// TwinCAT 3 PLC project MC3_Multi_IPC1
// ProgramVersion: 3.1.4026.13
// libraries:
//   Tc2_EtherCAT, * (Beckhoff Automation GmbH)
//   Tc2_Standard, * (Beckhoff Automation GmbH)
//   Tc2_System, * (Beckhoff Automation GmbH)
//   Tc2_Utilities, * (Beckhoff Automation GmbH)
//   Tc3_EventLogger, * (Beckhoff Automation GmbH)
//   Tc3_Mc3PlanarMotion, * (Beckhoff Automation GmbH)
//   Tc3_Module, * (Beckhoff Automation GmbH)
//   Tc3_Physics, * (Beckhoff Automation GmbH)
//   Tc3_XL_Motion, * (Beckhoff Automation GmbH)
//   Tc3_XtsInterface,newest,Beckhoff Automation GmbH
// project tree:
//   DUTs/ E_EcState.TcDUT (not stored), E_MergeMode.TcDUT (not stored), E_MergeType.TcDUT (not stored), E_SwitchOpMode.TcDUT (not stored), E_TrackNum.TcDUT, MoverSort.TcDUT (not stored), ST_Color_Code.TcDUT (not stored), ST_DivertConfig.TcDUT (not stored), ST_ExpMoverStatus.TcDUT (not stored), ST_MergeConfig.TcDUT (not stored), ST_MoverConfig.TcDUT (not stored), ST_PlanarTrackConfig.TcDUT (not stored), ST_SectorConfig.TcDUT (not stored), ST_ShortcutConfig.TcDUT (not stored), ST_StaticSectorStatus.TcDUT (not stored), ST_SwitchConfig.TcDUT (not stored), ST_SwitchStatus.TcDUT (not stored), ST_TrackConfig.TcDUT (not stored)
//   GVLs/ GVL_DataExchange.TcGVL, GVL_MC.TcGVL
//   / PlcTask.TcTTO (not stored)
//   POUs/ FB_PWM.TcPOU, FB_TrackObject.TcPOU, IsBetween.TcPOU (not stored), MAIN_S1.TcPOU, F_GetTrackEnum.TcPOU (not stored)
//   XlMover/DUTs/ DUT.TcDUT (not stored), ST_MoverInfo.TcDUT (not stored), ST_MoverOnTrackInfo.TcDUT
//   XlMover/ITFs/ I_Mover.TcIO
//   XlMover/POUs/ FB_Mover.TcPOU

// ---- DUTs/E_TrackNum.TcDUT
TYPE E_TrackNum :
{attribute 'qualified_only'}
{attribute 'strict'}
	(
	MainStart 	:= 1,	
	Big 		:= 2,
	MainEnd		:= 3,
	Small 		:= 4);	
END_TYPE

// ---- XlMover/DUTs/ST_MoverOnTrackInfo.TcDUT
TYPE ST_MoverOnTrackInfo :
STRUCT
	TargetPosition 		: LREAL;
	TargetTrack 		: Otcid;
	Remainingdistance 	: LREAL;
	Gap 				: LREAL;
	LimitV 				: LREAL;
	LimitA 				: LREAL;
	LimitD 				: LREAL;
	LimitJ 				: LREAL;
	GapMode				: MC.MC_GAP_MODE_ON_TRACK;
	DynamicMode			: MC.MC_DYNAMIC_MODE_ON_TRACK;
	Movementtype		: MC.MC_MOVEMENT_TYPE_ON_TRACK;
	
END_STRUCT
END_TYPE

// ---- GVLs/GVL_DataExchange.TcGVL
{attribute 'qualified_only'}
VAR_GLOBAL
	Dynamics AT%Q*: ST_Dynamics;
	Reset : BOOL;
	Run: BOOL;
	SafetyInRun : BOOL; 
	
	aMoverInfos : ARRAY[1..nNumMovers] OF ST_MoverInfo;
	
	
END_VAR

// ---- GVLs/GVL_MC.TcGVL

VAR_GLOBAL CONSTANT
	nNumMovers			: UINT := 12;
	nNumTracks			: UINT := 4;
	XtsShortcutOid				: otcid := 16#01010490 ;
	XtsOutterLoopOid 			: otcid := 16#01010480;
	
	fMagnetEntry : LREAL := 1766; //PLEASE ENTER THE MAGNET ENTRY!!!
	fMagnetExit : LREAL := 2332; //PLEASE ENTER THE MAGNET EXIT!!!
	
    standardAccel : LREAL := 4000; 
    standardDecel : LREAL :=4000; 
    standardJerk : LREAL := 16000; 

END_VAR
VAR_GLOBAL PERSISTENT
	nNumActiveMovers	: UINT := 1;
END_VAR	
VAR_GLOBAL
	

	fbXtsEnvironment			: 	FB_XtsEnvironment;
	ipXtsProcessingUnit			:   I_XtsProcessingUnit1;
	cmdFeedback					: 	XtsCommandFeedback;
	buffer						:   BYTE;
	
	fbMover						:	ARRAY[1..GVL_MC.nNumMovers] OF FB_Mover;
	iMover						:	ARRAY[1..GVL_MC.nNumMovers] OF I_Mover;
	aDynamics					:  	DynamicConstraint_PathXY;
	Feedback 					:	ARRAY[1..GVL_MC.nNumMovers] OF MC_PlanarFeedback;
	TrackFeedback 				:	ARRAY[1..GVL_MC.nNumTracks] OF MC_PlanarFeedback;
	aMcTracks					:	ARRAY[1..GVL_MC.nNumTracks] OF MC_PlanarTrack;
	ExitSystem 					: 	MC_PlanarTrackConnectionOut;
	EnterSystem 				:	MC_PlanarTrackConnectionIn;	
	Mover						:	ARRAY[0..GVL_MC.nNumMovers] OF MoverSort;
	defaultGap					:	LREAL := 900.0;
	SafetyOK			 AT %I* :	BOOL;
END_VAR

// ---- XlMover/ITFs/I_Mover.TcIO

INTERFACE I_Mover

METHOD CycleUpdate : BOOL
VAR_INPUT
END_VAR
END_METHOD

PROPERTY distToEndOfTrack : Lreal
GET
END_GET
END_PROPERTY

METHOD Init : BOOL
VAR_INPUT
	XtsMover:  I_XtsXlMover1;
	XtsProcessingUnit :  I_XtsProcessingUnit1;
END_VAR
END_METHOD

METHOD JoinNearestTrack : BOOL


VAR

END_VAR
END_METHOD

METHOD LeaveSystemAt : BOOL
VAR_INPUT
	ConnectionOut: REFERENCE TO MC_PlanarTrackConnectionOut;	
	gap : LREAL; 		
END_VAR
END_METHOD

METHOD MoveOnTrack : BOOL
VAR_INPUT
	track: REFERENCE TO MC_PlanarTrack;	
	targetPos: LREAL;
	gap : LREAL; 

END_VAR
END_METHOD

PROPERTY MoverStopped : BOOL
GET
END_GET
SET
END_SET
END_PROPERTY

PROPERTY P_Dynamics : REFERENCE TO DynamicConstraint_PathXY;
GET
END_GET
END_PROPERTY

PROPERTY P_IsInitialized : bool
GET
END_GET
END_PROPERTY

PROPERTY P_MoverOTCID : OTCID
GET
END_GET
SET
END_SET
END_PROPERTY

PROPERTY P_PlanarFeedback : REFERENCE TO MC_PlanarFeedback
GET
END_GET
END_PROPERTY

PROPERTY P_PlanarMover :   REFERENCE TO  MC_PlanarMover
GET
END_GET
END_PROPERTY

PROPERTY P_SyncFeedback :  REFERENCE TO MC_PlanarFeedbackGearInPosOnTrackWithMasterMover
GET
END_GET
END_PROPERTY

PROPERTY P_TargetTrack : UDINT
GET
END_GET
SET
END_SET
END_PROPERTY

PROPERTY Rework : BOOL
GET
END_GET
SET
END_SET
END_PROPERTY

METHOD SyncToOtherMover : Bool
VAR_INPUT
	masterSyncPos : LREAL; // Position on the master track
	followerSyncPos : LREAL; // position on the follower track
	PlanarMoverToFollow: REFERENCE TO Tc3_Mc3PlanarMotion.MC_PlanarMover;
	masterTrack : REFERENCE TO Tc3_Mc3PlanarMotion.MC_PlanarTrack; 
	followerTrack : REFERENCE TO Tc3_Mc3PlanarMotion.MC_PlanarTrack; 
	velo :  REFERENCE TO LREAL; 
END_VAR
END_METHOD

METHOD  UpdateXtsTrack
VAR_INPUT
END_VAR
VAR

END_VAR
END_METHOD

PROPERTY XlProcessingUnit : I_XtsProcessingUnit1
GET
END_GET
END_PROPERTY

PROPERTY XtsComFeed : REFERENCE TO  XtsCommandFeedback
GET
END_GET
END_PROPERTY

PROPERTY XtsXlMover :  I_XtsXlMover1
GET
END_GET
END_PROPERTY

END_INTERFACE

// ---- XlMover/POUs/FB_Mover.TcPOU
{attribute 'no_assign'}
FUNCTION_BLOCK FB_Mover IMPLEMENTS I_Mover
VAR_INPUT
END_VAR
VAR_OUTPUT
END_VAR
VAR
	_bIsInitialized: BOOL;	

	fbPlanarMover : MC_PlanarMover;
	fbPlanarFeedback: MC_PlanarFeedback;
	trackTrail: MC_PlanarTrackTrail;
	SyncMoverFeedback: Tc3_Mc3PlanarMotion.MC_PlanarFeedbackGearInPosOnTrackWithMasterMover;
	
	_GearInOptions: Tc3_Mc3PlanarMotion.ST_GearInPosOnTrackWithMasterMoverOptions;
	_stMoveOnTrackOptions: ST_MoveOnTrackOptions;
	_stLeaveSystemAtOptions : ST_LeaveSystemAtOptions;
	
	_syncTrail : MC_PlanarTrackTrail;
	
	CmdFeedback :  XtsCommandFeedback;
	ipXtsMover:   I_XtsXlMover1;
	ipXtsProcessingUnit:  I_XtsProcessingUnit1;

	_stMoverInfos : ST_MoverInfo;	
	_stMoverOnTrackInfos : MC_MOVER_ON_TRACK_INFORMATION;

	_nextMcTrackOid: OTCID;
	_stDynamics: DynamicConstraint_PathXY;
	_TargetTrack : UDINT;
	_ReWork : BOOL;
	_partConfig: UINT;
	_InSync :BOOL; 
	_PositionOnTrack : LREAL;
	_Track : OTCID; 
	_distToEndOfTrack : LREAL;

	fbResult						: FB_TcMessage;
	_ipComObject					: ITComObject;
	PID_OnTrackInfos				: PTCID := 16#05030180;
	bInit 							: BOOL;
END_VAR



METHOD CycleUpdate : BOOL
VAR_INPUT
END_VAR

VAR_INST
	_trackEnum: e_TrackNum;

END_VAR
IF NOT _bIsInitialized THEN
	RETURN;
END_IF

fbPlanarMover.GetTrackTrailInformation(trackTrail);
_PositionOnTrack := fbPlanarMover.MCTOPLC.SETONTRACK.SetPos;
IF fbPlanarMover.MCTOPLC.SETONTRACK.TrackOID<>0 THEN 
	_Track := fbPlanarMover.MCTOPLC.SETONTRACK.TrackOID;
	_trackEnum := F_GetTrackEnum(fbPlanarMover.MCTOPLC.SETONTRACK.TrackOID); 
	_distToEndOfTrack := GVL_Mc.aMCTracks[_trackEnum].GetLength()-_PositionOnTrack;
END_IF

fbPlanarMover.Update();
fbPlanarFeedback.Update();
SyncMoverFeedback.Update();

_stMoverinfos.MoverOtcid :=TO_STRING(fbPlanarMover.MCTOPLC.STD.MoverOID) ;
_stMoverinfos.IsActive := ipXtsMover.GetIsActive(0);
_stMoverinfos.ActPos :=  ipXtsMover.GetPositionInfo_trackPosition(0);
_stMoverinfos.ActVelo := fbPlanarMover.MCTOPLC.SETONTRACK.SetVelo;
_stMoverinfos.IsVirtuell := ipXtsMover.GetIsVirtualFeedbackEnabled(0);
_stMoverinfos.Positition :=	fbPlanarMover.MCTOPLC.SETONTRACK.SetPos;
_stMoverinfos.Track := TO_STRING(_trackEnum);
_stMoverinfos.Error := fbPlanarMover.Error;
_stMoverinfos.ErrorID := fbPlanarMover.ErrorId;
_stMoverinfos.PlanarMoverCommandMode :=  TO_STRING(fbPlanarMover.MCTOPLC.STD.CommandMode);
_stMoverinfos.State :=  TO_STRING(fbPlanarMover.MCTOPLC.STD.State);
_stMoverinfos.Gap := _stMoverOnTrackInfos.Gap;
_stMoverinfos.LimitAcc := _stMoverOnTrackInfos.LimitA;
_stMoverinfos.LimitDec := _stMoverOnTrackInfos.LimitD;
_stMoverinfos.LimitJerk := _stMoverOnTrackInfos.LimitJ;
_stMoverinfos.LimitVelo := _stMoverOnTrackInfos.LimitV;
_stMoverinfos.TargetTrackPosition := _stMoverOnTrackInfos.TargetPosition;
_stMoverinfos.TargetTrack := _stMoverOnTrackInfos.TargetTrack;
_stMoverinfos.RemainingDistance := _stMoverOnTrackInfos.Remainingdistance;




UpdateXtsTrack();
GetOnTrackInfos() ;
END_METHOD

PROPERTY distToEndOfTrack : Lreal
GET
distToEndOfTrack := _distToEndOfTrack;
END_GET
END_PROPERTY

METHOD GetComObject : BOOL
VAR_INPUT
	nObjectId: OTCID;
END_VAR
IF FW_ObjMgr_GetObjectInstance(	oid		:= nObjectId, 
								iid		:= TC_GLOBAL_IID_LIST.IID_ITComObject, 
								pipUnk	:= ADR(_ipComObject)) = 0
THEN
	GetComObject := TRUE;
END_IF
END_METHOD

METHOD GetOnTrackInfos : BOOL
VAR
	nData 			: UDINT := SIZEOF(MC_MOVER_ON_TRACK_INFORMATION);
	pData 			: PVOID := ADR(MC_MOVER_ON_TRACK_INFORMATION);
	stEventEntry	: TcEventEntry;
	pstEventEntry	: REFERENCE TO TcEventEntry REF= stEventEntry;
END_VAR
VAR_INST
	hResult : HRESULT;
	bError : BOOL;
END_VAR
bError := FALSE;

IF _ipComObject <> 0 THEN 
	 hResult := 	_ipComObject.TcgetObjPara(		pid := PID_OnTrackInfos,
													nData := nData,
													pData := pData,
													pgp := 0); 	
	IF hResult = 0 THEN
		GetOnTrackInfos := TRUE;
ELSE
	HRESULTAdsErr_TO_TcEventEntry(hResult,stEventEntry);
	IF NOT fbResult.EqualsToEventEntryEx( stOther := stEventEntry) THEN
		fbResult.CreateEx(stEventEntry, 0);
		fbResult.Send(0);
		fbResult.Release();
	END_IF
		bError := TRUE;
	END_IF							
END_IF
END_METHOD

METHOD Init : BOOL
VAR_INPUT

	XtsMover:   I_XtsXlMover1;
	XtsProcessingUnit :  I_XtsProcessingUnit1;
END_VAR



ipXtsMover:= XtsMover;
ipXtsProcessingUnit :=  XtsProcessingUnit;

_stMoveOnTrackOptions.direction := MC_Direction.mcDirectionPositive;
_stMoveOnTrackOptions.gapMode := MC_GAP_MODE_ON_TRACK.Fast1D;
_stMoveOnTrackOptions.gap:= 800;

_syncTrail.AddTrack(track:= GVL_Mc.aMCTracks[E_TrackNum.Small]); 
_syncTrail.AddTrack(track:= GVL_Mc.aMCTracks[E_TrackNum.MainStart]); 


//_stDynamics.SetValuesVADJ(500, 4000, 4000, 10000);




	_bIsInitialized := TRUE;
	Init := TRUE;

IF NOT bInit THEN
	IF GetComObject(nObjectId:=fbPlanarMover.MCTOPLC.STD.MoverOID) THEN
		bInit:=TRUE;
	END_IF
	RETURN;
END_IF
END_METHOD

METHOD JoinNearestTrack : BOOL


VAR_INST
	nForCounter: UINT;
	mcTrackOid: OTCID;
	partOid: OTCID;
	cmdFeedback					: 	XtsCommandFeedback;
	objectInfo: PlanarObjectInfo;
END_VAR
partOid := ipXtsMover.GetPositionInfo_partObjectId(cmdFeedback);

IF partOid = 0 THEN
	RETURN;
END_IF

IF cmdFeedback.IsDone THEN
	mcTrackOid := ipXtsProcessingUnit.XlPartWithOid(partOid, cmdFeedback).GetMcTrackOid(cmdFeedback);
	
	FOR nForCounter := 1 TO GVL_MC.nNumTracks DO
		objectInfo := GVL_MC.aMcTracks[nForCounter].GetPlanarObjectInfo();
		IF objectInfo.Id = mcTrackOid THEN
			fbPlanarMover.JoinTrack(fbPlanarFeedback, GVL_MC.aMcTracks[nForCounter], _stDynamics, 0); 
			RETURN;
		END_IF
	END_FOR
END_IF
END_METHOD

METHOD LeaveSystemAt : BOOL
VAR_INPUT
	ConnectionOut: REFERENCE TO MC_PlanarTrackConnectionOut;
	gap : LREAL; 
END_VAR
_stLeaveSystemAtOptions.gap := gap;
_stLeaveSystemAtOptions.gapMode := MC_GAP_MODE_ON_TRACK.Fast1D; 
_stLeaveSystemAtOptions.dynamicMode :=  MC_DYNAMIC_MODE_ON_TRACK.None;

fbPlanarMover.LeaveSystemAt(fbPlanarFeedback, ConnectionOut,  _stDynamics,_stLeaveSystemAtOptions);
END_METHOD

METHOD MoveOnTrack : BOOL
VAR_INPUT
	track: REFERENCE TO MC_PlanarTrack;	
	targetPos: LREAL;
	gap : LREAL; 
END_VAR
_stMoveonTrackOptions.gap := gap; 

fbPlanarMover.MoveOnTrack(
	commandFeedback:= fbPlanarFeedback, 
	targetTrack:= track, 
	targetPositionOnTrack:= targetPos, 
	constraint:= _stDynamics, 
	options:= _stMoveOnTrackOptions);
END_METHOD

PROPERTY MoverStopped : BOOL
GET
MoverStopped := (fbPlanarMover.MCTOPLC.SETONTRACK.SetVelo < 20);
END_GET
SET
END_SET
END_PROPERTY

PROPERTY P_Dynamics : REFERENCE TO DynamicConstraint_PathXY;
GET

P_Dynamics REF= _stDynamics;
END_GET
END_PROPERTY

PROPERTY P_IsInitialized : bool
GET
P_IsInitialized := _bIsInitialized;
END_GET
END_PROPERTY

PROPERTY P_MoveOnTrackOptions  : REFERENCE TO  ST_MoveOnTrackOptions
GET
P_MoveOnTrackOptions REF= _stMoveOnTrackOptions;
END_GET
END_PROPERTY

PROPERTY P_MoverInfos : REFERENCE TO ST_MoverInfo
GET
P_MoverInfos  REF= _stMoverInfos;
END_GET
END_PROPERTY

PROPERTY p_MoverOTCID : OTCID
GET
p_MoverOTCID := fbPlanarMover.MCTOPLC.STD.MoverOID;
END_GET
SET
END_SET
END_PROPERTY

PROPERTY P_PlanarFeedback : REFERENCE TO MC_PlanarFeedback
GET
P_PlanarFeedback REF= fbPlanarFeedback;
END_GET
END_PROPERTY

PROPERTY P_PlanarMover :   REFERENCE TO  MC_PlanarMover
GET
P_PlanarMover REF= fbPlanarMover;
END_GET
END_PROPERTY

PROPERTY P_SyncFeedback :  REFERENCE TO MC_PlanarFeedbackGearInPosOnTrackWithMasterMover
GET
P_SyncFeedback REF= SyncMoverFeedback;
END_GET
END_PROPERTY

PROPERTY P_TargetTrack : UDINT
GET
P_TargetTrack := _TargetTrack ;
END_GET
SET
_TargetTrack := P_TargetTrack;
END_SET
END_PROPERTY

PROPERTY Rework : BOOL
GET
Rework := _Rework;
END_GET
SET
_Rework := Rework;
END_SET
END_PROPERTY

METHOD SyncToOtherMover : BOOL
VAR_INPUT
	masterSyncPos : LREAL; // Position on the master track
	followerSyncPos : LREAL; // position on the follower track
	PlanarMoverToFollow: REFERENCE TO Tc3_Mc3PlanarMotion.MC_PlanarMover;
	masterTrack : REFERENCE TO Tc3_Mc3PlanarMotion.MC_PlanarTrack; 
	followerTrack : REFERENCE TO Tc3_Mc3PlanarMotion.MC_PlanarTrack; 
	velo : REFERENCE TO LREAL; 
END_VAR

VAR
	trail: Tc3_Mc3PlanarMotion.MC_PlanarTrackTrail;

END_VAR
_GearInOptions.allowedSlaveSyncDirections := MC_SYNC_DIRECTIONS.Positive; 
_GearInOptions.directionMasterSyncPosition := MC_DIRECTION.mcDirectionNonModulo; 
_GearInOptions.directionSlaveSyncPosition := MC_DIRECTION.mcDirectionNonModulo;  
_GearInOptions.followMover := FALSE; 
_GearInOptions.gap := 0; // elimnate gap funciton 
_GearInOptions.inSyncToleranceDistance :=0; 
_GearInOptions.moduloToleranceMasterSyncPosition := 0; 
_GearInOptions.moduloToleranceSlaveSyncPosition := 0;  
_stDynamics.V := velo; 

fbPlanarMover.GearInPosOnTrackWithMasterMover(
	commandFeedback:=  SyncMoverFeedback , 
	masterMover:= PlanarMoverToFollow , 
	trackTrail:= _syncTrail, // may need to give a trail maybe not
	masterSyncPosition:= masterSyncPos, 
	masterSyncPositionTrack:= MasterTrack , 
	slaveSyncPosition:= followerSyncPos, 
	slaveSyncPositionTrack:= followerTrack, 
	constraint:=_stDynamics , 
	options:=_GearInOptions );
END_METHOD

METHOD PUBLIC UpdateXtsTrack
VAR_INPUT
END_VAR
VAR_STAT
	nTrackCount: UINT;
	oid1: OTCID;
	oid2: OTCID;
	
	nForCounter: UINT;
	nPartConfigCount: UINT;
	
	partConfig1: OTCID;
	partConfig2: OTCID;
	
	mcTrackOid1: OTCID;
	mcTrackOid2: OTCID;
	trackOid: OTCID;
	
	nTrackTrailCount: UDINT;
	actTrackOid: OTCID;
	nIndexInTrail: UDINT;
END_VAR
nTrackTrailCount := trackTrail.TrackCount;
actTrackOid := fbPlanarMover.MCTOPLC.SETONTRACK.TrackOID;

IF nTrackTrailCount <= 1 THEN
	RETURN;
END_IF

FOR nForCounter := 1 TO UDINT_TO_UINT(nTrackTrailCount) DO
	oid1 := trackTrail.GetTrackOidAt(nForCounter);
	IF oid1 = actTrackOid THEN
		IF nForCounter < nTrackTrailCount THEN
			oid2 := trackTrail.GetTrackOidAt(nForCounter + 1);
			EXIT;
		ELSE
			RETURN; //last one ine track trail
		END_IF
	END_IF
END_FOR

IF oid2 = _nextMcTrackOid AND ipXtsMover.GetPositionInfo_partPosition(CmdFeedback) < 600 THEN //no change
	RETURN;
END_IF

nTrackCount := ipXtsProcessingUnit.TrackCount();

FOR nForCounter := 1 TO nTrackCount DO
	nPartConfigCount := ipXtsProcessingUnit.Track(nForCounter, CmdFeedback).PartConfigCount(); 
	
	IF nPartConfigCount >= 2  THEN
		partConfig1 := ipXtsProcessingUnit.Track(nForCounter, CmdFeedback).GetPartConfigOidAt(1, 0);
		partConfig2 := ipXtsProcessingUnit.Track(nForCounter, CmdFeedback).GetPartConfigOidAt(2, 0);
//
		
		IF partConfig1 = 0 OR partConfig2 = 0 THEN
			CONTINUE;
		END_IF
		
		mcTrackOid1 := ipXtsProcessingUnit.XlPartWithOid(partConfig1, CmdFeedback).GetMcTrackOid(0);
		mcTrackOid2 := ipXtsProcessingUnit.XlPartWithOid(partConfig2, CmdFeedback).GetMcTrackOid(0);
		IF mcTrackOid1 = oid1 AND mcTrackOid2 = oid2   THEN
			trackOid := ipXtsProcessingUnit.Track(nForCounter, CmdFeedback).GetObjectId();
			ipXtsMover.SetActiveTrackObjectId(trackOid, CmdFeedback);
			
			IF CmdFeedback.IsDone THEN
				_nextMcTrackOid := oid2;
			END_IF
			
			RETURN;
		END_IF
	END_IF
END_FOR
END_METHOD

PROPERTY XlProcessingUnit : I_XtsProcessingUnit1
GET
XlProcessingUnit := ipXtsProcessingUnit;
END_GET
END_PROPERTY

PROPERTY XtsComFeed : REFERENCE TO  XtsCommandFeedback
GET
XtsComFeed REF= CmdFeedback;
END_GET
END_PROPERTY

PROPERTY XtsXlMover : I_XtsXlMover1
GET
XtsXlMover := ipXtsMover;
END_GET
END_PROPERTY

END_FUNCTION_BLOCK

// ---- POUs/FB_PWM.TcPOU
FUNCTION_BLOCK FB_PWM
VAR_INPUT
	SafeetyOk : BOOL;
	Torque: INT;
END_VAR

VAR
  	ModuleState AT %I* : UINT;
	
 	Control AT %Q* :  UINT;
 	TargetTorque AT %Q*: INT; 	

 	State  : INT := 1;
 	PwmTimer : ton;
END_VAR

VAR_OUTPUT
	Ready : BOOL;
END_VAR


Ready := FALSE;
CASE State OF 

	1:
		IF SafeetyOk THEN
			State := 2;
		END_IF
	2: 
		Control := 6;
		IF ModuleState = 40 OR ModuleState = 33 THEN
			State := 5;
		END_IF
	5:
		Control := 128;
		IF ModuleState = 96 OR ModuleState = 33 OR ModuleState = 168 THEN
			State := 10;
		END_IF
	10:
		Control := 6;
		IF ModuleState = 33 THEN
			state := 15;
		END_IF	
	15:
		Control := 7;
		IF ModuleState = 35 OR ModuleState = 163 or ModuleState = 2083 THEN
			State := 20;
		END_IF	
	20:	
		Control := 15;
		IF ModuleState = 4135 OR ModuleState = 4263THEN
			state := 25;
		END_IF
	24:
	  //IF Torque = 0  THEN
			State := 25;
	//	END_IF	
		PwmTimer(in := FALSE,PT := T#30S);
	25:
		IF ModuleState = 40 THEN
			State := 5;
		END_IF
		Ready := TRUE;
		
		IF Torque > 0 THEN
			TargetTorque := Torque ;
		ELSIF Torque = 0 AND TargetTorque > 0  THEN	
			TargetTorque :=  TargetTorque - REAL_TO_INT((INT_TO_REAL(TargetTorque)*0.07));
		END_IF	
		
		PwmTimer(in := TargetTorque > 300,PT := T#30S);
		IF PwmTimer.Q  THEN
			PwmTimer(in := FALSE,PT := T#30S);
			State := 35;
		END_IF 
	35:
		IF TargetTorque >0 THEN
			TargetTorque := TargetTorque -4;
		ELSIF 	TargetTorque = 0  THEN
				State := 24;
		END_IF	

END_CASE

END_FUNCTION_BLOCK

// ---- POUs/FB_TrackObject.TcPOU
FUNCTION_BLOCK FB_TrackObject
// for a track/part this block keeps a list of the movers in order with their positions on a track

VAR_INPUT
	TrackID: OTCID;
	iMover	:REFERENCE TO ARRAY[1..nNumMovers] OF I_Mover;
	trackLength : LREAL;// this should be a loookup but I don't know how to look it up so I'm going to pass it externally 
END_VAR

VAR_OUTPUT
	bBusy: BOOL;
	bDone: BOOL;
	bError: BOOL;
	bInit: BOOL;
	ipResultMessage: I_TcMessage := fbResult;
	moverIDs : ARRAY[1..nNumMovers] OF UDINT;
END_VAR

VAR
	nNumMoversThisTrack: UDINT; //numberofMovers currently on this track
	nMoverList: ARRAY [1..nNumMovers] OF OTCID; //list of movers currently on the track 

	distToNextMover : ARRAY[1..nNumMovers] OF LREAL;  
END_VAR

VAR

	fbResult: FB_TcMessage;
	_ipComObject: ITComObject;
	PID_MOverList				: PTCID := 16#05030149;
	PID_NumMover				: PTCID := 16#050300C5;
END_VAR

IF NOT bInit THEN
	IF GetComObject(nObjectId:=TrackID) THEN
		bInit:=TRUE;
	END_IF
	RETURN;
END_IF

METHOD CyclicUpdate : BOOL
VAR_INPUT
END_VAR

VAR
	J: UDINT;
	I: UDINT;
END_VAR
IF bInit THEN 
	GetNumMovers(); 
	GetMoverList(); 
END_IF 
MEMSET(ADR(moverIDs),0,SIZEOF(moverIDs)); // have to clear the list 
FOR J := 1 TO nNumMoversThisTrack DO  
	FOR I := 1 TO nNumMovers DO  
		IF iMover[I].P_MoverOTCID = nMoverList[J] THEN 
			moverIDs[J] := I; 
		END_IF
	END_FOR
END_FOR
FOR I := 1 TO nNumMoversThisTrack DO 
	IF I <= nNumMoversThisTrack -1 THEN
		distToNextMover[I] := fbMover[moverIDs[I+1]].distToEndOfTrack - fbMover[moverIDs[I]].distToEndOfTrack;
	ELSIF I = nNumMoversThisTrack THEN
		distToNextMover[I] := trackLength - fbMover[moverIDs[I]].distToEndOfTrack;
	END_IF
END_FOR
END_METHOD

METHOD findMergePosition : BOOL
VAR_INPUT
	mergeSyncCommandPos : LREAL;
	spaceToMerge :LREAL; 
END_VAR
VAR_OUTPUT 
	nMoverToFollow: UDINT; 
	mergeWithoutFollow : BOOL; 
	mergeNotPossible : BOOL; 
END_VAR
VAR_INST 
	I: UDINT;
	moverInMerge: UDINT;
END_VAR
mergeNotPossible := TRUE; 
mergeWithoutFollow:=FALSE;
nMoverToFollow := 0; 
moverInMerge := 0;
// do not get fancy,  go through the list find all the distances between
//cyclic update finds builds a list of moers on the track and their spaceing 

IF nNumMoversThisTrack = 0  THEN // if there's no movers on the track we can just merge 
	mergeWithoutFollow := TRUE;
	mergeNotPossible := FALSE; 
ELSE
	// find a mover to follow starting at sync position look for a space to merge sized hole 
	FOR I := 1 TO nNumMoversThisTrack DO 
		IF fbMover[moverIDs[I]].distToEndOfTrack > mergeSyncCommandPos THEN // this mover is a potentialmover to follow 
			IF distToNextMover[I] > spaceToMerge THEN // follow this mover 
				nMoverToFollow := moverIDs[I]; //yes follow this mover 
				mergeNotPossible := FALSE; // the merge is possible 
				EXIT ; //get out of the loop we want the first one 
			END_IF
		END_IF
	END_FOR 
END_IF
IF mergeNotPossible THEN 
	nMoverToFollow := 0; 
END_IF
END_METHOD

METHOD GetComObject : BOOL
VAR_INPUT
	nObjectId: OTCID;
END_VAR
IF FW_ObjMgr_GetObjectInstance(	oid		:= nObjectId, 
								iid		:= TC_GLOBAL_IID_LIST.IID_ITComObject, 
								pipUnk	:= ADR(_ipComObject)) = 0
THEN
	GetComObject := TRUE;
END_IF
END_METHOD

METHOD GetMoverList : BOOL
VAR
	nData 			: UDINT := SIZEOF(nMoverList);
	pData 			: PVOID := ADR(nMoverList);
	stEventEntry	: TcEventEntry;
	pstEventEntry	: REFERENCE TO TcEventEntry REF= stEventEntry;
END_VAR
VAR_INST
	hResult : HRESULT;
END_VAR
bError := FALSE;

IF _ipComObject <> 0 THEN 
	 hResult := 	_ipComObject.TcgetObjPara(		pid := PID_MOverList,
													nData := nData,
													pData := pData,
													pgp := 0); 	
	IF hResult = 0 THEN
		GetMoverList := TRUE;
	ELSE
		HRESULTAdsErr_TO_TcEventEntry(hResult,stEventEntry);
		IF NOT fbResult.EqualsToEventEntryEx( stOther := stEventEntry) THEN
			fbResult.CreateEx(stEventEntry, 0);
			fbResult.Send(0);
			fbResult.Release();
		END_IF
		bError := TRUE;
	END_IF							
END_IF
END_METHOD

METHOD GetNumMovers : BOOL
VAR
	stEventEntry: TcEventEntry;
	pstEventEntry: REFERENCE TO TcEventEntry := stEventEntry;
	nData 			: UDINT := SIZEOF(nNumMoversThisTrack);
	pData 			: PVOID := ADR(nNumMoversThisTrack);
END_VAR

VAR_INST
	hResult : HRESULT;
END_VAR
bError := FALSE;

IF _ipComObject <> 0 THEN 	
	nData := SIZEOF(nNumMoversThisTrack);
	pData  := ADR(nNumMoversThisTrack);

	 hResult := 	_ipComObject.TcGetObjPara(		pid := PID_NumMover,
													nData := nData,
													pData := pData,
													pgp := 0); 	
													
	IF hResult = 0 THEN
		GetNumMovers := TRUE;
	ELSE
		HRESULTAdsErr_TO_TcEventEntry(hResult,stEventEntry);
		IF NOT fbResult.EqualsToEventEntryEx( stOther := stEventEntry) THEN
			fbResult.CreateEx(stEventEntry, 0);
			fbResult.Send(0);
			fbResult.Release();
		END_IF
		bError := TRUE;
	END_IF							
END_IF
END_METHOD

END_FUNCTION_BLOCK

// ---- POUs/MAIN_S1.TcPOU
PROGRAM MAIN_S1

VAR
	voltage_trafo	 	AT %I* 	: REAL ;
	current_trafo		AT %I* 	: REAL;  
	power_trafo					: REAL;

	b110SyncState AT %I* :UINT ;
	b110State AT %I* :UINT;  
	EtherCATWCState23To49 AT %I* : BOOL; 
	EtherCATWCState50To76 AT %I* : BOOL; 
	AktiveSystem : BOOL := TRUE;
	bSwitch : BOOL := TRUE;
	nState: UINT;
	MoverState :ARRAY[1..GVL_MC.nNumMovers] OF UINT;
	nForCounter ,i: UINT;
	Velo : LREAL := 2000;
	fbPWM : FB_PWM;
	//mover :ARRAY[1..nNumMovers] OF MC_PlanarMover;
	
	LocalSystemTime : FB_LocalSystemTime;
	
	fbTrackobject : FB_TrackObject;

	ipXlMover: 	I_XtsXlMover1;


	state : INT := -1;
	arrivedOTCID : OTCID;
	Start :BOOL;
	bAlldone : BOOL;
	
	

	test : otcid; 
	XPU_Number : UINT := 1; 	
	
	Short : BOOL := TRUE;
	
	XtsOutterLoopOid: OTCID ;	
	XtsShortcutOid: OTCID ;
	
	Init : BOOL ; 
	EndTrack : INT := E_TrackNum.MainEnd;
 	StartTrack : INT :=E_TrackNum.MainStart ;
	MoverNo : DINT;
	SystemReady: BOOL;
	IsDetectionOnStartupEnabled : BOOL := FALSE;
	
	MagnetValue AT%Q*: INT;
	bMagnetOn : BOOL;	
	Fault : BOOL;
	SwitchCurrent :lreal := 7;
	Switchcounter : DINT;
	FP_Counter : r_trig;
	

	aMoverTrack : ARRAY[1..GVL_Mc.nNumMovers] OF otcid;
	FirstMoverTrackPos : LREAL;
	MoverGap : LREAL;
	FTrigTrackCount : F_Trig;
	MoverNo1  : UDINT;
	gapStart: LREAL := 5600;
	gapLength: LREAL := 2000;
	moverInFront: UDINT;
	mover1FollowDist: LREAL;
	followSyncPos: LREAL;
	masterSyncPos: LREAL;
	masterPosAtSync: LREAL;
	followerPosAtSync: LREAL;
	endOfBigTrack : LREAL; 
     endOfSmallTrack : LREAL; 
     endOfMainTrack : LREAL; 
     followerToEndOfTrack: LREAL;
     leaderToEndofTrack: LREAL;
     distToMoverInFront: LREAL;
     vara: Tc3_Mc3PlanarMotion.PlanarObjectInfo;
  
     getList: BOOL;
     directMerge: BOOL;
     mergeNotPossible: BOOL;

	A : LREAL := 0.63;
	B : LREAL := 0.21;
	C : LREAL := 10;
	
	cmdFeedback: Tc3_XtsInterface.XtsCommandFeedback;
	BUFFER: BYTE;
	
	xReset AT %Q*: BOOL;
	xStart AT %Q*: BOOL;
	EtherCATFault: BOOL;
	syncFault: BOOL;

	
	haltDynamics : DynamicConstraint_PathXY;
	stMoverConfigSlow	: ST_MoverConfig;
	stMoverConfigNormal : ST_MoverConfig;
	stMoverConfigFast  : ST_MoverConfig;
	stMoverCfgAggressive : ST_MoverConfig;
	stMoverCfgHalt : ST_MoverConfig;
	MoverStopDone : BOOL;
	
	Fp_error : R_trig;
	
	ModuleState1 AT%I*: E_EcState;
	ModuleState2 AT%I*: E_EcState;
	ModuleState3 AT%I*: ARRAY[0..2] OF E_EcState;
	
	MessageTrigger : ARRAY[1..20] OF R_trig;
	
	
	TestPowerMat : BOOL := TRUE;
	StopTime : TIME := T#1S;
	StopTimer :ARRAY[1..nNumMovers] OF ton;
	StartTimer :ARRAY[1..nNumMovers] OF BOOL;
	SwitchParkPos : LREAL := 3500;
	trapError: BOOL;
	trapErrorID: UDINT;
	moverWithFault: UDINT;
	stepWithFault: INT;
	stopAndWait : ARRAY[1..nNumMovers] OF TON; 
	
	AllDone : BOOL;
	InitDone  :BOOL;
END_VAR


VAR_INPUT
	remoteState AT %I*: INT;
END_VAR


// =====================
// Initalize XTS Utility
GVL_MC.fbXtsEnvironment.Init(GVL_MC.cmdFeedback);
IF NOT GVL_MC.cmdFeedback.IsDone THEN
	RETURN;
END_IF


//=================== Check State of Modules===========================================
IF EtherCATWCState23To49 OR EtherCATWCState50To76 THEN 
	EtherCATFault := TRUE; 
END_IF
IF b110SyncState <> 1 THEN 
	syncFault := TRUE;  
END_IF

MessageTrigger[1](clk:=ModuleState1 <> 8 AND state> 0);
IF MessageTrigger[1].Q THEN
	ADSLOGSTR(msgCtrlMask:= ADSLOG_MSGTYPE_LOG , msgFmtStr:= 'Module Fault Line 1 %s' , strArg:= TO_STRING(ModuleState1));
END_IF

MessageTrigger[2](clk:=ModuleState2 <> 8 AND state> 0);
IF MessageTrigger[2].Q THEN
	ADSLOGSTR(msgCtrlMask:= ADSLOG_MSGTYPE_LOG , msgFmtStr:= 'Module Fault Line 2 %s ' , strArg:= TO_STRING(ModuleState2));
END_IF

MessageTrigger[3](clk:=ModuleState3[0] <> 8 AND state> 0);
IF MessageTrigger[3].Q THEN
	ADSLOGSTR(msgCtrlMask:= ADSLOG_MSGTYPE_LOG , msgFmtStr:= 'Module Fault Line 3 Default SyncUnit %s ' , strArg:= TO_STRING(ModuleState3[0]));
END_IF

MessageTrigger[4](clk:=ModuleState3[1] <> 8 AND state> 0);
IF MessageTrigger[4].Q THEN
	ADSLOGSTR(msgCtrlMask:= ADSLOG_MSGTYPE_LOG , msgFmtStr:= 'Module Fault Line 3 XtsTask SyncUnit %s ' , strArg:= TO_STRING(ModuleState3[1]));
END_IF

MessageTrigger[5](clk:=ModuleState3[2] <> 8 AND state> 0);
IF MessageTrigger[5].Q THEN
	ADSLOGSTR(msgCtrlMask:= ADSLOG_MSGTYPE_LOG , msgFmtStr:= 'Module Fault Line 3 PlcTask SyncUnit %s ' , strArg:= TO_STRING(ModuleState3[2]));
END_IF


//===========================================================================================

GVL_MC.ipXtsProcessingUnit :=  GVL_MC.fbXtsEnvironment.ProcessingUnit(XPU_Number,0);
AllDone  := TRUE;
FOR i := 1 TO GVL_MC.nNumMovers DO 	
	
	IF NOT InitDone  THEN
		ipXlMover  :=  GVL_MC.fbXtsEnvironment.ProcessingUnit(XPU_Number, 0).XlMover(i, 0);
		AllDone := AllDone AND GVL_MC.fbMover[i].Init(ipXlMover, GVL_MC.ipXtsProcessingUnit); 
	END_IF
	
	
	Fp_error(clk := GVL_MC.fbMover[i].P_PlanarMover.Error AND GVL_MC.fbMover[i].XtsXlMover.GetIsActive(0) AND state = 100);
	IF Fp_error.Q AND FALSE THEN
		state := 140;
		Fault := TRUE;

		ADSLOGSTR(msgCtrlMask:= ADSLOG_MSGTYPE_LOG , msgFmtStr:= 'Mover %s Faulted ' , strArg:= INT_TO_STRING(i));
	ELSE
		Fault := FALSE;
	END_IF
	


	GVL_MC.Feedback[i].Update();
	GVL_MC.fbMover[i].CycleUpdate();
	GVL_MC.iMover[i] := GVL_MC.fbMover[i];

	GVL_MC.fbMover[i].P_Dynamics.SetValuesVADJ(stMoverConfigNormal.Velo,stMoverConfigNormal.Accel, stMoverConfigNormal.Decel, stMoverConfigNormal.Jerk);

	GVL_MC.fbMover[i].P_MoveOnTrackOptions.gap := 900;
	GVL_MC.fbMover[i].P_MoveOnTrackOptions.direction := MC_Direction.mcDirectionPositive;
	GVL_MC.fbMover[i].P_MoveOnTrackOptions.gapMode := MC_GAP_MODE_ON_TRACK.Fast1D;
	GVL_DataExchange.aMoverInfos[i] :=  GVL_MC.fbMover[i].P_MoverInfos;
END_FOR	

IF AllDone THEN
	InitDone := TRUE;
ELSE 
	RETURN;
END_IF
GVL_DataExchange.Dynamics.v := stMoverConfigNormal.Velo;
GVL_DataExchange.Dynamics.A := stMoverConfigNormal.Accel;
GVL_DataExchange.Dynamics.D := stMoverConfigNormal.Decel;
GVL_DataExchange.Dynamics.J := stMoverConfigNormal.Jerk;

fbTrackobject(TrackID:= GVL_mc.aMcTracks[E_TrackNum.big].MCTOPLC_STD.TrackOID,iMover:= gvl_mc.iMover ); 
fbTrackobject.CyclicUpdate();

FOR i := 1 TO GVL_MC.nNumTracks DO 
	GVL_MC.aMcTracks[i].Update();
	GVL_MC.TrackFeedback[i].Update();
END_FOR	








IF state < 99 AND xReset THEN 
	IF State = 1 THEN 
		xReset := FALSE; 
	END_IF 
	state := 0; 
END_IF
IF state = 99 AND xStart AND remoteState  = 99 THEN   
	state := 100;  
END_IF

CASE state OF
	0: 
		
		FOR i := 1 TO GVL_MC.nNumTracks DO  
			GVL_MC.aMcTracks[i].Enable(GVL_MC.TrackFeedback[i]);
			state := 1;
		END_FOR
		
	1: 	
		bAlldone := TRUE;
		FOR i := 1 TO GVL_MC.nNumTracks DO  
			bAlldone := bAlldone AND GVL_MC.aMcTracks[i].MCTOPLC_STD.State = MC_PLANAR_STATE.Enabled ;
		END_FOR

 		IF bAlldone THEN
			state := 2;
		END_IF

	2:	
	
		FOR i := 1+GVL_MC.nNumActiveMovers TO GVL_MC.nNumMovers DO  
			GVL_MC.fbMover[i].XlProcessingUnit.XlMover(i,0).SetStartupTrackPosition(0.2,0);	
			GVL_MC.fbMover[i].XlProcessingUnit.XlMover(i,0).SetIsVirtualFeedbackEnabled(1,0);
			GVL_MC.fbMover[i].XlProcessingUnit.XlMover(i,0).TriggerArrive(0);
		END_FOR
		IF  GVL_MC.nNumActiveMovers > 0 THEN
			FOR i :=1  TO GVL_MC.nNumActiveMovers DO 	
				GVL_MC.fbMover[i].XlProcessingUnit.XlMover(i,0).SetIsVirtualFeedbackEnabled(0,0);
			END_FOR 
		END_IF			
		state := 3;
		
	3:
		FOR i := 1 TO GVL_MC.fbXtsEnvironment.ProcessingUnit(1, 0).XlPartCount() DO
			 GVL_MC.fbXtsEnvironment.ProcessingUnit(1, 0).XlPart(i, 0).TriggerReset(0);
		END_FOR
		
		state := 5;
		
	5: 

		
		IF AktiveSystem THEN
			state := 10;
		ELSE
			state := 100;
		END_IF	

	10:
		FOR i := 1 TO GVL_MC.nNumActiveMovers DO
			GVL_MC.fbMover[i].P_PlanarMover.Reset(0);			
		END_FOR
		state := 11; 
	11:
		FOR i := 1 TO GVL_MC.nNumActiveMovers DO
			GVL_MC.fbMover[i].P_PlanarMover.Enable(0);		
		END_FOR
		state := 15;	
	15:
		bAlldone := TRUE;
		FOR i := 1 TO GVL_MC.nNumActiveMovers DO  
			bAlldone := bAlldone AND GVL_MC.fbMover[i].P_PlanarMover.MCTOPLC.STD.State = MC_PLANAR_STATE.Enabled ;	
		END_FOR
		
		IF bAlldone THEN
			state := 18;
		END_IF
	18: 
	
		FOR i := 1 TO GVL_MC.nNumActiveMovers DO  
			GVL_MC.fbMover[i].JoinNearestTrack(aMcTracks,nNumTracks);
			//set Sync trail=================================================	
			GVL_MC.fbMover[i].ClearSyncTrail();
			GVL_MC.fbMover[i].SetSyncTrail(aMcTracks[E_TrackNum.Small]);
			GVL_MC.fbMover[i].SetSyncTrail(aMcTracks[E_TrackNum.MainEnd]);
			//===============================================================
		END_FOR
		state := 20;
	
	20:
		bAlldone := TRUE;
		FOR i := 1 TO GVL_MC.nNumActiveMovers DO  
			bAlldone := bAlldone AND GVL_MC.fbMover[i].fbPlanarMover.MCTOPLC.STD.CommandMode = MC_PLANAR_MOVER_COMMAND_MODE.OnTrack  ;	
			MoverState[i] := 10;
			
		END_FOR

		IF bAlldone THEN
			state := 99;
			Fault := FALSE;
		END_IF
		
	99:
	 	IF GVL_MC.nNumActiveMovers = 0 THEN
			state := 100;
		END_IF
		
	100: 
		arrivedOTCID := GVL_MC.EnterSystem.PopFirstMoverInQueue();
		IF arrivedOTCID <> 0 THEN
			FOR i := 1  TO GVL_MC.nNumMovers DO
				IF GVL_MC.fbMover[i].P_MoverOTCID = arrivedOTCID THEN
					MoverState[i] := 0;
				END_IF
			END_FOR
		END_IF
	
		FOR i := 1 TO GVL_MC.nNumMovers DO 
			
			IF MoverNo1 <> 0 AND_THEN GVL_MC.fbMover[MoverNo1].P_PlanarMover.MCTOPLC.SETONTRACK.TrackOID =  GVL_MC.aMcTracks[E_TrackNum.Big].MCTOPLC_STD.TrackOID THEN
				Short := FALSE;
			END_IF	
		
			CASE MoverState[i] OF 
			0:		 
				IF  bSwitch AND GVL_MC.fbMover[i].P_PlanarMover.MCTOPLC.SETONTRACK.TrackOID = GVL_MC.aMcTracks[E_TrackNum.MainStart].MCTOPLC_STD.TrackOID    THEN
					IF NOT short   THEN
						GVL_MC.fbMover[i].MoveOnTrack(GVL_MC.aMcTracks[E_TrackNum.Small], SwitchParkPos(* GVL_MC.aMcTracks[E_TrackNum.Small].GetLength()/2*), GVL_MC.defaultGap);
						MoverNo1 := i;
						Short := TRUE;
						MoverState[i] := 4;
					ELSE
						GVL_MC.fbMover[i].MoveOnTrack(GVL_MC.aMcTracks[E_TrackNum.Big],(GVL_MC.aMcTracks[E_TrackNum.Big].GetLength()-12000), GVL_MC.defaultGap);			
						MoverState[i] := 10;
					END_IF
				ELSIF NOT bSwitch AND  GVL_MC.fbMover[i].P_PlanarMover.MCTOPLC.SETONTRACK.TrackOID = GVL_MC.aMcTracks[E_TrackNum.MainStart].MCTOPLC_STD.TrackOID THEN
					GVL_MC.fbMover[i].MoveOnTrack(GVL_MC.aMcTracks[EndTrack],GVL_MC.aMcTracks[EndTrack].GetLength()-450, GVL_MC.defaultGap);
					MoverState[i] := 12;				
				END_IF
			4:
				IF fbMover[i].P_PlanarFeedback.Error AND NOT trapError THEN //trap the error once.   
						trapError := fbMover[i].P_PlanarFeedback.Error; 
						trapErrorID := fbMover[i].P_PlanarFeedback.ErrorId;
						stepWithFault := 4;
 						moverWithFault := i; 
					END_IF
					IF fbMover[i].P_PlanarFeedback.Done THEN 
						MoverState[i] := 5; //50;
						stopAndWait[i](IN:=TRUE, PT:=StopTime); 
					END_IF 	
			5:
				stopAndWait[i](); 
					IF stopAndWait[i].Q  OR NOT TestPowerMat THEN // send the mover to a sync Position 2.6m before the end of the track 
						stopAndWait[i](IN:=FALSE); 							
						MoverState[i] := 6; 
					END_IF 	
				
			6:
               
                fbTrackobject.findMergePosition(
                   mergeSyncCommandPos := gapStart , 
                   spaceToMerge := gapLength, 
                   nMoverToFollow => moverInFront, 
                   mergeWithoutFollow => directMerge, 
                   mergeNotPossible => mergeNotPossible); 
								
                IF (directMerge OR moverInFront <> 0) AND NOT mergeNotPossible THEN
                                MoverState[i] := 7;
                END_IF 
			7:  //merge with gap zero
					//issue commmand to sync 
					IF  directMerge THEN 
						GVL_MC.fbMover[i].P_Dynamics.SetValuesVADJ(stMoverConfigNormal.velo,stMoverConfigNormal.Accel,stMoverConfigNormal.Decel,stMoverConfigNormal.Jerk);
						fbMover[i].MoveOnTrack(track:= GVL_Mc.aMCTracks[E_TrackNum.MainEnd], targetPos:= GVL_Mc.aMCtracks[E_TrackNum.Mainend].GetLength()-500, gap:= GVL_MC.defaultGap);

						MoverState[i] := 10; 
					ELSIF moverInFront <>0 THEN 
						fbMover[i].P_Dynamics.SetValuesVADJ(stMoverConfigNormal.velo,stMoverConfigNormal.Accel,stMoverConfigNormal.Decel,stMoverConfigNormal.Jerk);
						masterSyncPos := GVL_Mc.aMCTracks[E_TrackNum.Big].GetLength()-2500;
						masterPosAtSync := Mover[moverInFront].MoverPos; 
						followSyncPos := GVL_Mc.aMCTracks[E_TrackNum.Small].GetLength()- GVL_MC.defaultGap -2500;
						followerPosAtSync :=Mover[nForCounter].MoverPos; 
						fbMover[i].SyncToOtherMover( 
							masterSyncPos := masterSyncPos,
							masterTrack := GVL_Mc.aMCTracks[E_TrackNum.Big],
							followerSyncPos := followSyncPos,
							followerTrack := GVL_Mc.aMCTracks[e_TrackNum.Small],
							PlanarMoverToFollow := fbMover[moverInFront].P_PlanarMover,
							velo:= stMoverConfigNormal.velo);
							MoverState[i] := 8; 
						// reduce the gap of the leading mover 
						fbMover[moverInFront].MoveOnTrack(track:= GVL_Mc.aMcTracks[E_TrackNum.MainEnd], targetPos:= GVL_Mc.aMcTracks[E_TrackNum.MainEnd].GetLength()-250, gap:= 0);

					END_IF 
			
  			
                  
  			8: // wait for in Sync 
                  IF Gvl_mc.fbMover[i].P_SyncFeedback.Active AND  gvl_mc.MOver[moverInFront].TrackID =  GVL_Mc.aMCTracks[E_TrackNum.Big].MCTOPLC_STD.TrackOID THEN // actively syncing calculate distance from mover 
                  		
						followerToEndOfTrack := endOfSmallTrack - gvl_mc.Mover[i].MoverPos; 
                  		leaderToEndofTrack := endOfBigTrack - gvl_mc.Mover[moverInFront].MoverPos; 
                  		distToMoverInFront := followerToEndOfTrack - leaderToEndofTrack; 
						
                  ELSE 
                 		followerToEndOfTrack := 0; 
                 		leaderToEndofTrack := 0; 
                 		distToMoverInFront := 0;
                  END_IF
				  
               	IF fbMover[nForCounter].P_SyncFeedback.inSync OR  MOver[nForCounter].TrackID =  GVL_Mc.aMCTracks[E_TrackNum.MainEnd].MCTOPLC_STD.TrackOID THEN 
						MoverState[i] := 10;
						Short :=FALSE;
				ELSIF	fbMover[nForCounter].P_SyncFeedback.Error THEN
						MoverState[i] := 6;
				END_IF 

			10:

				IF  (  GVL_MC.fbMover[i].P_PlanarMover.MCTOPLC.SETONTRACK.SetPos > 500 AND GVL_MC.fbMover[i].P_PlanarMover.MCTOPLC.SETONTRACK.TrackOID <>  GVL_MC.aMcTracks[StartTrack].MCTOPLC_STD.TrackOID) THEN
					GVL_MC.fbMover[i].MoveOnTrack(GVL_MC.aMcTracks[EndTrack], GVL_MC.aMcTracks[EndTrack].GetLength()- 200, GVL_MC.defaultGap);
					MoverState[i] := 12;
				END_IF
		
			12: 
				//500mm after that the boundary change commmand is issued 
				IF SystemReady AND GVL_MC.fbMover[i].P_PlanarMover.MCTOPLC.SETONTRACK.SetPos > GVL_MC.aMcTracks[E_TrackNum.MainEnd].GetLength() - 2300 AND // 2300
				(GVL_MC.fbMover[i].P_PlanarMover.MCTOPLC.SETONTRACK.TrackOID = GVL_MC.aMcTracks[E_TrackNum.MainEnd].MCTOPLC_STD.TrackOID)  THEN 
					GVL_MC.fbMover[i].LeaveSystemAt(GVL_MC.ExitSystem, GVL_MC.defaultGap); 
					MoverState[i] := 15; 
				END_IF
				
			15:
			 	IF GVL_MC.fbMover[i].XlProcessingUnit.XlMover(i,0).GetIsVirtualFeedbackEnabled(0) AND //In some cases the planar mover gots an error, we have to evaluate why
					GVL_MC.fbMover[i].P_PlanarMover.Error THEN
					GVL_MC.fbMover[i].P_PlanarMover.Reset(0);
					MoverState[i] := 16; 
				END_IF
				
			16: 
				GVL_MC.fbMover[i].P_PlanarMover.Disable(0);
				MoverState[i] := 17; 
		
			END_CASE
		END_FOR	
		
		140:
			FOR i := 1 TO GVL_MC.nNumMovers DO  
				GVL_MC.fbMover[i].P_PlanarMover.Halt(GVL_MC.Feedback[i], haltDynamics);
			END_FOR	
			
				state := 145;
			
		145:
			bAllDone := TRUE;
				FOR i := 1 TO GVL_MC.nNumMovers DO  
				IF NOT(GVL_MC.Feedback[i].Done OR GVL_MC.Feedback[i].Error) THEN
					bAllDone := FALSE;
					EXIT;
				END_IF
			END_FOR
			
			IF bAllDone THEN
				state := 150;
			END_IF
		
		//Disable
		150:
			MoverStopDone := TRUE;
			FOR i := 1 TO GVL_MC.nNumMovers DO  
					GVL_MC.fbMover[i].P_PlanarMover.Disable(GVL_MC.Feedback[i]);
			END_FOR
				
			state := 0;
		
		
	
END_CASE

bMagnetOn := FALSE;
FOR nForCounter:=1 TO GVL_MC.nNumMovers DO
	IF  GVL_MC.fbMover[nForCounter].XtsXlMover.GetPositionInfo_trackObjectId(0) = GVL_mc.XtsShortcutOid AND (IsBetween(GVL_MC.fbMover[nForCounter].XtsXlMover.GetPositionInfo_trackPosition(0), gvl_mc.fMagnetEntry - (Velo*0.06), gvl_mc.fMagnetExit(*- (Velo*0.04)*))) THEN
		bMagnetOn := TRUE;
	END_IF
END_FOR


SwitchCurrent := ((A*(((Velo/1000)*(Velo/1000))))+(B*(Velo/1000))+C);
IF bMagnetOn AND NOT Fault THEN
	MagnetValue := TO_INT(SwitchCurrent*1310);
ELSE
 	MagnetValue := 0;
END_IF

FP_Counter(clk:=bMagnetOn);

IF FP_Counter.Q THEN
	Switchcounter := Switchcounter+1;

END_IF

//distanceMonitoring of Mover 1 when on the big track 
IF GVL_MC.Mover[1].TrackID = GVL_Mc.aMcTracks[E_TrackNum.MainStart].MCTOPLC_STD.TrackOID THEN //calculate out how far it is to the mover in front 
	IF GVL_MC.Mover[moverInFront].MoverPos -  GVL_Mc.Mover[1].MoverPos > 10 THEN 
		mover1FollowDist := GVL_Mc.Mover[moverInFront].MoverPos -  GVL_Mc.Mover[1].MoverPos;
	END_IF   
END_IF



// Calculation of the transformator power 
power_trafo := voltage_trafo * current_trafo;

END_PROGRAM
